SUBAPPLICATION Uebung_070c_AUI (* WBSD auf UT ausgeben (Adapter Version) *)
  (* Standard: 61499-2; Description: Copyright (c) 2023 Meisterschulen am Ostbahnhof This program and the accompanying materials are made available under the terms of the Eclipse Public License 2.0 which is available at https://www.eclipse.org/legal/epl-2.0/ SPDX-License-Identifier: EPL-2.0 *)
  (* Version 1.0, 2026-06-01, Franz Höpfinger, Meisterschulen am Ostbahnhof, WBSD mit Compound Scaling (Adapter Version) *)
  PACKAGE Uebungen;
  IMPORT Uebungen::const::UT::TECU::DefaultPool_TECU_Numeric::NumberVariable_Wheel_based_machine_speed_N;
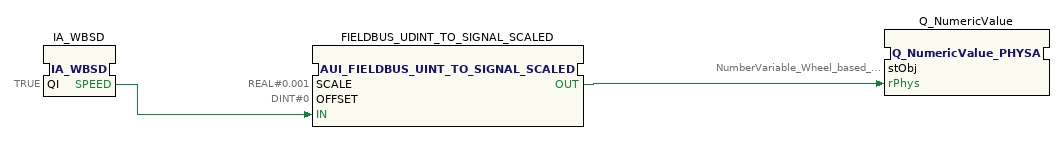
  FBS
    IA_WBSD : isobus::tecu::IA_WBSD(QI := TRUE);
    FIELDBUS_UDINT_TO_SIGNAL_SCALED : logiBUS::signalprocessing::fieldbus::AUI_FIELDBUS_UINT_TO_SIGNAL_SCALED(SCALE := REAL#0.001, OFFSET := DINT#0);
    Q_NumericValue : isobus::UT::Q::Q_NumericValue_PHYSA(stObj := NumberVariable_Wheel_based_machine_speed_N);
  END_FBS
  ADAPTER_CONNECTIONS
    FIELDBUS_UDINT_TO_SIGNAL_SCALED.OUT TO Q_NumericValue.rPhys;
    IA_WBSD.SPEED TO FIELDBUS_UDINT_TO_SIGNAL_SCALED.IN;
  END_CONNECTIONS
END_SUBAPPLICATION
